// TIA Portal V18 export
FUNCTION_BLOCK "SlewDec"   // FB123, LAD
TITLE = SlewInc
{ S7_Optimized_Access := 'TRUE' }
// Written BY Kristopher Gimenez Feb 17th ,2023
// This block will be used to slew the output but the at the set rate per second base on input slew rate
// stored: AutoNumber false, MemoryReserve 100, SetENOAutomatically false
   VAR_INPUT
      SlewRate : Real;   // Slew rate in mA/sec
   END_VAR
   VAR_IN_OUT
      RealValue : Real;
   END_VAR
   VAR
      Slew : Bool;
      Dec_TON : TON_TIME;
   END_VAR
   VAR_TEMP
      tempReal : Real;
   END_VAR
BEGIN

REGION Network 1: Slew rate in mA/sec
   // Decrease the input value by the slew rate
   // Decreasing every 10ms divide rate by 100
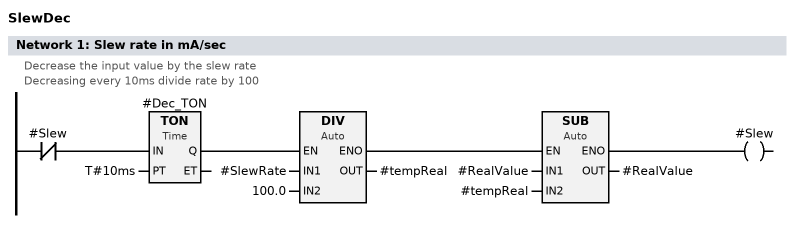
   RUNG wire#powerrail
      I_Contact( #Slew )
      { S7_Templates := "time_type := Time" } #Dec_TON.TON(pt := T#10ms, et =>)
      Div(in1 := #SlewRate, in2 := 100.0, out => #tempReal)
      Sub(in1 := #RealValue, in2 := #tempReal, out => #RealValue)
      Coil( #Slew )
   END_RUNG
   // the same network as SCL:
   #Dec_TON(IN := NOT #Slew, PT := T#10ms);   // TON
   IF #Dec_TON.Q THEN
       #tempReal := #SlewRate / 100.0;
       #RealValue := #RealValue - #tempReal;
   END_IF;
   #Slew := #Dec_TON.Q;
END_REGION
END_FUNCTION_BLOCK
